// FB Controle/FB_PAlloc
(*
    ════════════════════════════════════════════════════════════════
    FB_PAlloc - Alocador de Potência Ativa (PRIORIDADE MÁXIMA)
    ════════════════════════════════════════════════════════════════
*)
FUNCTION_BLOCK FB_PAlloc
VAR_INPUT
    P_total_cmd_kW : REAL;          // Comando de P total (do FB_PI)
END_VAR

VAR_OUTPUT
    P_allocated_kW : REAL;          // ✅ ADICIONAR ESTA SAÍDA!
END_VAR

VAR
    i : UINT;
    P_target_i : REAL;
    P_actual_i : REAL;
    P_total_calc : REAL;
    proportion : REAL;
END_VAR


P_total_calc := 0.0;

FOR i := 1 TO Global.NMAXINVERSORES DO     
    
    IF GVL_Persis.InvActivePower[i] > 0.0 THEN
        
        // Proporção do inversor
        proportion := GVL_Persis.InvActivePower[i] / Global.InstalledPower;
        
        // P proporcional
        P_target_i := P_total_cmd_kW * proportion;
        
        // Limita apenas pela nominal (ignora S_max por enquanto)
        P_actual_i := MIN(P_target_i, GVL_Persis.InvActivePower[i]);
        
        // Armazena P
        Global.P_inv_kW[i] := P_actual_i;
        
        // Setpoint percentual
        IF GVL_Persis.InvActivePower[i] > 0.0 THEN
            Global.P_inv_Percent[i] := (P_actual_i / GVL_Persis.InvActivePower[i]) * 100.0;
        ELSE
            Global.P_inv_Percent[i] := 0.0;
        END_IF
        
        P_total_calc := P_total_calc + P_actual_i;
        
    ELSE
        Global.P_inv_kW[i] := 0.0;
        Global.P_inv_Percent[i] := 0.0;
    END_IF
    
END_FOR

// ✅ ATUALIZA SAÍDA
P_allocated_kW := P_total_calc;

END_FUNCTION_BLOCK

// FB Controle/FB_PI
FUNCTION_BLOCK FB_PI
VAR_INPUT
    setpoint    : REAL;         		// Setpoint desejado
    feedback    : REAL;         		// Medição atual (feedback)
    Kp          : REAL;         		// Ganho proporcional
    Ki          : REAL;         		// Ganho integral
    OutMax      : REAL;         		// Limite superior de saída
    OutMin      : REAL;         		// Limite inferior de saída
    CycleTime   : REAL;         		// Tempo de ciclo (s)
    RampUp      : REAL := 1.0E+6;  		//  Rampa de subida (unidade/s). Default = sem limite
    RampDown    : REAL := 1.0E+6;  		//  Rampa de descida (unidade/s). Default = sem limite
    Deadband    : REAL := 0.0;          //  deadband em kW (já convertido de %)
    bReset      : BOOL := FALSE;        //  reset do PI
END_VAR

VAR_OUTPUT
    u           : REAL;         		// Saída do controlador
    erro        : REAL;         		// Erro atual (setpoint - feedback)
    bSaturated  : BOOL;         		// TRUE = saída saturada
END_VAR

VAR
    integ           : REAL := 0.0;      // Integral acumulada
    LastOut         : REAL := 0.0;
    erroAtual       : REAL;             // Erro no ciclo atual
    u_prop          : REAL;             // Componente proporcional
    u_raw           : REAL;             // Saída antes da saturação
    u_limited       : REAL;         	// Saída após saturação, antes da rampa
    delta           : REAL;         	// Variação desejada
    delta_max       : REAL;         	// Variação máxima permitida
    primeiro_ciclo  : BOOL := TRUE;     // Flag de primeira execução
    sinal_saturacao : INT;              // +1: saturado max, -1: saturado min, 0: não saturado
END_VAR


// ════════════════════════════════════════════════════════════════
// Reset explícito
// ════════════════════════════════════════════════════════════════
IF bReset THEN
    integ := 0.0;
    LastOut := 0.0;
    u := 0.0;
    bSaturated := FALSE;
    primeiro_ciclo := TRUE;
    RETURN;
END_IF

// ════════════════════════════════════════════════════════════════
// Inicialização suave na primeira execução
// ════════════════════════════════════════════════════════════════
IF primeiro_ciclo THEN
    integ := 0.0;
    primeiro_ciclo := FALSE;
    
    // Se quiser inicializar LastOut com valor atual do medidor:
    // LastOut := feedback;  // Opcional: evita salto inicial
END_IF

// ════════════════════════════════════════════════════════════════
// Cálculo do Erro + Deadband
// ════════════════════════════════════════════════════════════════
erroAtual := setpoint - feedback;

// ✅ Deadband
IF ABS(erroAtual) < Deadband THEN
    erroAtual := 0.0;
END_IF

erro := erroAtual;  // Saída para diagnóstico

// ════════════════════════════════════════════════════════════════
// Componente Proporcional
// ════════════════════════════════════════════════════════════════
u_prop := Kp * erroAtual;

// ════════════════════════════════════════════════════════════════
// Saída Raw (P + I + LastOut)
// ══════════════════════════════════════════���═════════════════════
u_prop := Kp * erroAtual;
u_raw := u_prop + integ;

// ════════════════════════════════════════════════════════════════
// Saturação
// ════════════════════════════════════════════════════════════════
IF u_raw > OutMax THEN
    u_limited := OutMax;
    bSaturated := TRUE;
    sinal_saturacao := 1;
ELSIF u_raw < OutMin THEN
    u_limited := OutMin;
    bSaturated := TRUE;
    sinal_saturacao := -1;
ELSE
    u_limited := u_raw;
    bSaturated := FALSE;
    sinal_saturacao := 0;
END_IF

// ════════════════════════════════════════���═══════════════════════
// Rate Limiter (Rampa)
// ════════════════════════════════════════════════════════════════
delta := u_limited - LastOut;

IF delta > 0.0 THEN
    delta_max := RampUp * CycleTime;
    IF delta > delta_max THEN
        u := LastOut + delta_max;
    ELSE
        u := u_limited;
    END_IF
ELSIF delta < 0.0 THEN
    delta_max := RampDown * CycleTime;
    IF ABS(delta) > delta_max THEN
        u := LastOut - delta_max;
    ELSE
        u := u_limited;
    END_IF
ELSE
    u := u_limited;
END_IF
// ════════════════════════════════════════════════════════════════
// Anti-windup Melhorado (Conditional Integration)
// ════════════════════════════════════════════════════════════════
// Regras:
// 1. NÃO saturado → acumula normalmente
// 2. Saturado MAS erro na direção oposta → permite desacumular
// 3. Saturado E erro na mesma direção → freeze (não acumula)

IF NOT bSaturated THEN
    // Caso 1: Normal - acumula integral
    integ := integ + (Ki * erroAtual * CycleTime);
    
ELSIF (sinal_saturacao = 1 AND erroAtual < 0.0) OR (sinal_saturacao = -1 AND erroAtual > 0.0) THEN
    // Caso 2: Saturado MAS erro está tentando sair da saturação
    // Permite acumular para ajudar a desaturar
    integ := integ + (Ki * erroAtual * CycleTime);
    
ELSE
    // Caso 3: Saturado E erro empurrando mais para saturação
    // NÃO acumula (freeze integral)
    // integ permanece inalterado
END_IF

// ════════════════════════════════════════════════════════════════
// Atualiza LastOut
// ════════════════════════════════════════════════════════════════
LastOut := u;

END_FUNCTION_BLOCK

// FB Controle/FB_Diagnostico
(*
    ════════════════════════════════════════════════════════════════
    FB_Diagnostico - Diagnóstico de Fator de Potência
    ════════════════════════════════════════════════════════════════
    
    Gera diagnóstico completo do sistema de compensação de PF,
    incluindo alarmes, recomendações e estatísticas.
    
    ═══���════════════════════════════════════════════════════════════
*)

FUNCTION_BLOCK FB_Diagnostico
VAR_INPUT
    P_allocated_kW : REAL;
    Q_commanded_kvar : REAL;
    Q_allocated_kvar : REAL;
    Q_capacity_kvar : REAL;
    PF_measured : REAL;
    PF_achieved : REAL;
    bQ_limited : BOOL;
END_VAR

VAR
    Q_deficit : REAL;
    Q_deficit_pct : REAL;
    S_total_avail : REAL;
    S_total_used : REAL;
    bank_size : REAL;
    bank_size_int : DINT;  // ✅ DINT (não INT)
END_VAR

// ════════════════════════════════════════════════════════════════
// 1. ARMAZENA VALORES BÁSICOS
// ════════════════════════════════════════════════════════════════

Global.P_generated_kW := P_allocated_kW;
Global.P_allocated_kW := P_allocated_kW;
Global.Q_commanded_kvar := Q_commanded_kvar;
Global.Q_allocated_kvar := Q_allocated_kvar;
Global.Q_available_kvar := Q_capacity_kvar;
Global.PF_measured := PF_measured;
Global.PF_achieved := PF_achieved;

// Q medido (do ponto de conexão)
Global.Q_measured_kvar := Global.Qt;  // Já convertido em kvar pelo FB_AjustaLeitura

// ════════════════════════════════════════════════════════════════
// 2. CALCULA DÉFICIT DE Q
// ════════════════════════════════════════════════════════════════

Q_deficit := Q_commanded_kvar - Q_allocated_kvar;
Global.Q_deficit_kvar := Q_deficit;

// Déficit percentual
IF ABS(Q_commanded_kvar) > 0.1 THEN
    Q_deficit_pct := (ABS(Q_deficit) / ABS(Q_commanded_kvar)) * 100.0;
ELSE
    Q_deficit_pct := 0.0;
END_IF
Global.Q_deficit_percent := Q_deficit_pct;

// ════════════════════════════════════════════════════════════════
// 3. CALCULA UTILIZAÇÃO DE S
// ════════════════════════════════════════════════════════════════

// S total disponível
S_total_avail := Global.InstalledSmax;
Global.S_total_available_kVA := S_total_avail;

// S total usado
S_total_used := SQRT((P_allocated_kW * P_allocated_kW) + (Q_allocated_kvar * Q_allocated_kvar));
Global.S_total_used_kVA := S_total_used;

// Utilização percentual
IF S_total_avail > 0.0 THEN
    Global.S_utilization_pct := (S_total_used / S_total_avail) * 100.0;
ELSE
    Global.S_utilization_pct := 0.0;
END_IF

// ════════════════════════════════════════════════════════════════
// 4. CALCULA UTILIZAÇÃO DE Q
// ════════════════════════════════════════════════════════════════

Global.Q_capacity_total_kvar := Q_capacity_kvar;

IF Q_capacity_kvar > 0.0 THEN
    Global.Q_utilization_pct := (ABS(Q_allocated_kvar) / Q_capacity_kvar) * 100.0;
ELSE
    Global.Q_utilization_pct := 0.0;
END_IF

// ════════════════════════════════════════════════════════════════
// 5. CALCULA TAMANHO DE BANCO DE CAPACITORES
// ════════════════════════════════════════════════════════════════

IF Q_deficit > 0.1 THEN
    // Adiciona 10% de margem
    bank_size := ABS(Q_deficit) * 1.1;
	bank_size := DINT_TO_REAL(TRUNC(bank_size / 5.0) + 1) * 5.0;
    Global.Capacitor_bank_size_kvar := bank_size;
    Global.Capacitor_bank_recommended := TRUE;
ELSE
    Global.Capacitor_bank_size_kvar := 0.0;
    Global.Capacitor_bank_recommended := FALSE;
END_IF

// ════════════════════════════════════════════════════════════════
// 6. DETERMINA STATUS DE PF
// ════════════════════════════════════════════════════════════════

IF PF_achieved >= Global.PF_target THEN
    Global.PF_OK := TRUE;
    Global.PFErro := FALSE;
    Global.PF_alarm_code := 0;  // OK
    Global.PF_alarm_message := 'Fator de Potencia OK';
ELSE
    Global.PF_OK := FALSE;
    
    IF bQ_limited THEN
        Global.PFErro := TRUE;
        
        // Classifica severidade
        IF Q_deficit_pct > 20.0 THEN
            Global.PF_alarm_code := 2;  // Crítico
            Global.PF_alarm_message := 'CRITICO: Limite de Q atingido - Banco de capacitores necessario';
        ELSE
            Global.PF_alarm_code := 1;  // Aviso
            Global.PF_alarm_message := 'AVISO: Limite de Q atingido - Considerar banco de capacitores';
        END_IF
    ELSE
        // PF < 0.92 mas não por limite de Q (transitório)
        Global.PFErro := FALSE;
        Global.PF_alarm_code := 1;
        Global.PF_alarm_message := 'PF abaixo do alvo - Sistema compensando';
    END_IF
END_IF

// ════════════════════════════════════════════════════════════════
// 7. ATUALIZA HISTÓRICO (OPCIONAL - implementar com timers)
// ════════════════════════════════════════════════════════════════

// Atualiza PF mínimo
IF PF_achieved < Global.PF_min_24h THEN
    Global.PF_min_24h := PF_achieved;
END_IF

// Atualiza déficit máximo
IF Q_deficit > Global.Q_deficit_max_24h THEN
    Global.Q_deficit_max_24h := Q_deficit;
END_IF

// Conta alarmes (incrementar quando alarme dispara pela primeira vez)
// (Implementar com edge detection)

END_FUNCTION_BLOCK

// FB Controle/FB_PowerController
(*
    ════════════════════════════════════════════════════════════════
    FB_PowerController - Controlador de Potência Ativa
    ════════════════════════════════════════════════════════════════
    
    Responsabilidade:
    - Calcular comando de P (PI + Safety Margin + Limites de Fase)
    - Encapsular toda lógica relacionada a potência ativa
    
    Pipeline:
    1. PI → P_cmd_raw
    2. Safety Margin → P_cmd_with_margin
    3. Limitador de Fase → P_cmd_limited
    
    ════════════════════════════════════════════════════════════════
*)
FUNCTION_BLOCK FB_PowerController
VAR_INPUT
    ExportLimit_kW : REAL;      // Do scheduler (kW)
    Feedback_kW : REAL;         // Leitura do medidor (kW)
    bReset : BOOL;              // Reset do PI
END_VAR

VAR_OUTPUT
    P_cmd_kW : REAL;            // Comando final (kW)
    bSaturated : BOOL;          // PI saturado
    bPhase_limited : BOOL;      // Limitado por fase
    sLimited_phase : STRING;    // Qual fase limitou
    Margin_applied_kW : REAL;   // Margem aplicada (telemetria)
	EffectiveExportLimit_kW : REAL;
END_VAR

VAR
    // Sub-blocos
    fbPI : FB_PI;
    fbSafetyMargin : FB_SafetyMargin;
    fbFLimiter : FB_FLimiter;
	fbDroop : FB_DroopP;
    
    // Variáveis internas
    P_setpoint : REAL;
    P_cmd_raw : REAL;
    P_cmd_with_margin : REAL;
	lastInstalledPower : REAL := -1.0;
	
	// Droop
    P_error_kW : REAL;
    P_droop_kW : REAL;
	
    P_droop_max_kW : REAL;
    P_cmd_sum : REAL;
	
	// ✅ Deadband em kW (convertido de %)
	Deadband_P_kW     : REAL;
    Droop_Deadband_kW : REAL;
END_VAR

// ────────────────────────────────────────────────────────────────
// ETAPA 1: CONTROLADOR PI
// ────────────────────────────────────────────────────────────────

// Setpoint negativo (exportação)
P_setpoint := -ABS(ExportLimit_kW);

// Erro (kW)
P_error_kW := Feedback_kW - P_setpoint;

// Converte deadband (%) para kW (mínimo 1 kW)
// Recalcula apenas se InstalledPower mudou
IF lastInstalledPower <> Global.InstalledPower THEN
    Deadband_P_kW := MAX(1.0, Global.InstalledPower * (GVL_Persis.Deadband_P / 100.0));
    Droop_Deadband_kW := MAX(1.0, Global.InstalledPower * (GVL_Persis.Deadband_Droop / 100.0));
	Deadband_P_kW := MIN(20.0, MAX(1.0, Global.InstalledPower * (GVL_Persis.Deadband_P / 100.0)));
	Droop_Deadband_kW := MIN(20.0, MAX(1.0, Global.InstalledPower * (GVL_Persis.Deadband_Droop / 100.0)));		
    lastInstalledPower := Global.InstalledPower;
END_IF

// Limite máximo do droop (fração da potência instalada)
P_droop_max_kW := GVL_Persis.Droop_Max * Global.InstalledPower;

// Calcula droop
fbDroop(
    Enable      := GVL_Persis.Droop_Enable,
    bReset      := bReset,                 
    Error_kW    := P_error_kW,
    K_droop     := GVL_Persis.K_Droop,
    Deadband_kW := Droop_Deadband_kW,
    P_max_kW    := P_droop_max_kW
);

P_droop_kW := fbDroop.P_droop_kW;

// PI de potência ativa
fbPI(
    setpoint    := P_error_kW,
    feedback    := 0.0,
    Kp          := GVL_Persis.Kp_P,
    Ki          := GVL_Persis.Ki_P,
    OutMax      := Global.InstalledPower,
    OutMin      := 0.0,
    CycleTime   := Global.ControlCycle,
	RampUp      := GVL_Persis.RampUp_P,     
    RampDown    := GVL_Persis.RampDown_P,    
    Deadband    := Deadband_P_kW,
	bReset      := bReset          
);

// Soma droop + PI
P_cmd_sum := P_droop_kW + fbPI.u;

// Comando bruto (segue fluxo normal)
P_cmd_raw := P_cmd_sum;
IF P_cmd_raw < 0.0 THEN
    P_cmd_raw := 0.0;
ELSIF P_cmd_raw > Global.InstalledPower THEN
    P_cmd_raw := Global.InstalledPower;
END_IF
bSaturated := fbPI.bSaturated;

// ─────────────────────────────────────────���──────────────────────
// ETAPA 2: SAFETY MARGIN
// ────────────────────────────────────────────────────────────────

fbSafetyMargin(
    P_cmd_raw_kW := P_cmd_raw,
    Margin_pct := GVL_Persis.SafetyMargin_pct,
    TC_Power_kW := GVL_Persis.TC_Power_kW
);

P_cmd_with_margin := fbSafetyMargin.P_cmd_adjusted_kW;
Margin_applied_kW := fbSafetyMargin.Margin_applied_kW;  // ✅ Telemetria
EffectiveExportLimit_kW := P_setpoint + Margin_applied_kW;
// ────────────────────────────────────────────────────────────────
// ETAPA 3: LIMITADOR DE FASE
// ────────────────────────────────────────────────────────────────

fbFLimiter(
    P_cmd_in := P_cmd_with_margin,
    PowerMode := GVL_Persis.PowerMode
);

P_cmd_kW := fbFLimiter.P_cmd_out;
bPhase_limited := fbFLimiter.bPhase_limited;
sLimited_phase := fbFLimiter.sLimited_phase;

// ────────────────────────────────────────────────────────────────
// PROTEÇÃO FINAL: Potência Instalada
// ────────────────────────────────────────────────────────────────

IF P_cmd_kW > Global.InstalledPower THEN
    P_cmd_kW := Global.InstalledPower;
    bSaturated := TRUE;
END_IF

END_FUNCTION_BLOCK

// FB Controle/FB_SafetyMargin
(*
    ════════════════════════════════════════════════════════════════
    FB_SafetyMargin - Margem de Segurança para Correção de TC
    ════════════════════════════════════════════════════════════════
    
    Função:
    - Aplica margem de segurança para compensar erro de TC em baixas correntes
    - Desloca setpoint para lado da importação (garante não exportar)
    
    Exemplo:
    - P_cmd = 100 kW
    - TC_Power = 329 kW
    - Margin = 3%
    - SafetyMargin = 3% × 329 = 9.87 kW
    - P_adjusted = 100 - 9.87 = 90.13 kW
    ════════════════════════════════════════════════════════════════
*)
FUNCTION_BLOCK FB_SafetyMargin
VAR_INPUT
    P_cmd_raw_kW : REAL;        // Comando sem margem
    Margin_pct : REAL;          // Percentual (ex: 3.0)
    TC_Power_kW : REAL;         // Potência do TC
END_VAR

VAR_OUTPUT
    P_cmd_adjusted_kW : REAL;   // Comando com margem
    Margin_applied_kW : REAL;   // Margem aplicada (para telemetria)
END_VAR

VAR
    SafetyMargin_kW : REAL;
END_VAR

// ════════════════════════════════════════════════════════════════
// IMPLEMENTAÇÃO
// ════════════════════════════════════════════════════════════════
// 1. Proteção: se TC não configurado, não aplica margem
IF TC_Power_kW <= 0.0 THEN
    P_cmd_adjusted_kW := P_cmd_raw_kW;
    Margin_applied_kW := 0.0;
    RETURN;
END_IF

// 2. Calcula margem em kW
SafetyMargin_kW := (Margin_pct / 100.0) * TC_Power_kW;

// 3. Aplica margem (reduz comando)
P_cmd_adjusted_kW := P_cmd_raw_kW - SafetyMargin_kW;

// 4. Limita para não ficar negativo
IF P_cmd_adjusted_kW < 0.0 THEN
    P_cmd_adjusted_kW := 0.0;
END_IF

// 5. Armazena margem aplicada (para HMI)
Margin_applied_kW := SafetyMargin_kW;

END_FUNCTION_BLOCK

// FB Controle/FB_FLimiter
(*
    FB_FLimiter - Limitador por Fase
    
    Função:
    - Verifica se o comando causaria EXPORTAÇÃO excessiva em alguma fase
    - Se fase está IMPORTANDO: ignora (não há problema)
    - Se fase está EXPORTANDO: verifica se comando excederia limite
    
    Lógica:
    1. Calcula P futuro por fase = P_atual + (P_cmd / 3)
    2. Para cada fase EXPORTANDO (P < 0):
       - Verifica se P_futuro < P_phase_limit (mais exportação que permitido)
       - Se sim, calcula comando máximo para essa fase
    3. Usa o MENOR comando máximo entre as fases
    
    Convenção de sinais:
    - P > 0: Importação
    - P < 0: Exportação
    - MaxExportLimit: VALOR POSITIVO na agenda (ex: 90 kW)
    - P_phase_limit: NEGATIVO internamente (ex: -30 kW)
	    
    Exemplo:
    - Agenda: MaxExportLimit = 90 kW (sem sinal)
    - Internamente: P_phase_limit = -90/3 = -30 kW por fase
    - Se Pa = -25 kW (exportando 25 kW)
    - Se P_cmd = -18 kW (quer aumentar exportação)
    - P_future_A = -25 + (-18/3) = -31 kW → EXCEDE -30 kW → LIMITA
*)

FUNCTION_BLOCK FB_FLimiter
VAR_INPUT
    P_cmd_in : REAL;                // Comando de P calculado pelo PI (kW)
    PowerMode : UINT;               // 0=Total, 1=Por fase, 2=Ambos
END_VAR

VAR_OUTPUT
    P_cmd_out : REAL;               // Comando de P limitado por fase (kW)
    bPhase_limited : BOOL;          // TRUE = alguma fase limitou
	sLimited_phase : STRING;        // Qual fase limitou: 'A', 'B', 'C', 'AB', etc.
END_VAR

VAR
    P_cmd_per_phase : REAL;         // Comando adicional por fase (kW)
    P_future_A : REAL;              // P futuro na fase A após aplicar comando (kW)
    P_future_B : REAL;              // P futuro na fase B após aplicar comando (kW)
    P_future_C : REAL;              // P futuro na fase C após aplicar comando (kW)
    P_phase_limit : REAL;           // Limite de exportação por fase (kW negativo)
    P_max_cmd_A : REAL;             // Comando máximo permitido para fase A (kW)
    P_max_cmd_B : REAL;             // Comando máximo permitido para fase B (kW)
    P_max_cmd_C : REAL;             // Comando máximo permitido para fase C (kW)
    P_max_cmd_total : REAL;         // Comando máximo total permitido (kW)
	NO_LIMIT : REAL;                // Constante para "sem limite"
    bLimitA : BOOL;                 // Fase A está limitando
    bLimitB : BOOL;                 // Fase B está limitando
    bLimitC : BOOL;                 // Fase C está limitando
END_VAR

// Comando adicional por fase (distribuído equilibradamente)
P_cmd_per_phase := P_cmd_in / 3.0;

// Limite de exportação por fase
// Se MaxExportLimit = -90 kW, então por fase = -30 kW
P_phase_limit := -ABS(Global.MaxExportLimit) / 3.0;

// ════════════════════════════════════════════════════════════════
// ════════════════════════════════════════════════════════════════
// Inicialização
// ════════════════════════════════════════════════════════════════
NO_LIMIT := Global.InstalledPower * 10.0;  // Valor grande, mas realista
sLimited_phase := '';
bLimitA := FALSE;
bLimitB := FALSE;
bLimitC := FALSE;

// ════════════════════════════════════════════════════════════════
// Se PowerMode = 0, não verifica fase
// ════════════════════════════════════════════════════════════════
IF PowerMode = 0 THEN
    P_cmd_out := P_cmd_in;
    bPhase_limited := FALSE;
    RETURN;
END_IF

// ════════════════════════════════════════════════════════════════
// Proteção: Se InstalledPower não configurado
// ════════════════════════════════════════════════════════════════
IF Global.InstalledPower <= 0.0 THEN
    P_cmd_out := 0.0;
    bPhase_limited := TRUE;
    sLimited_phase := 'ERROR: InstalledPower=0';
    RETURN;
END_IF

// ════════════════════════════════════════════════════════════════
// Calcula P futuro em cada fase após aplicar comando
// ════════════════════════════════════════════════════════════════
P_future_A := Global.Pa + P_cmd_per_phase;
P_future_B := Global.Pb + P_cmd_per_phase;
P_future_C := Global.Pc + P_cmd_per_phase;

// ════════════════════════════════════════════════════════════════
// Verifica FASE A
// ════════════════════════════════════════════════════════════════
IF P_future_A < 0.0 THEN
    // Fase A estará EXPORTANDO após aplicar comando
    
    IF P_future_A < P_phase_limit THEN
        // Excederia o limite de exportação!
        // Calcula quanto PODE aumentar exportação sem exceder:
        // P_max_per_phase = P_limit - P_atual
        // P_max_total = P_max_per_phase * 3
        P_max_cmd_A := (P_phase_limit - Global.Pa) * 3.0;
        bLimitA := TRUE;
    ELSE
        // Dentro do limite: sem restrição
        P_max_cmd_A := NO_LIMIT;
    END_IF
    
ELSE
    // Fase A estará IMPORTANDO: sem problema
    P_max_cmd_A := NO_LIMIT;
END_IF

// ════════════════════════════════════════════════════════════════
// Verifica FASE B
// ════════════════════════════════════════════════════════════════
IF P_future_B < 0.0 THEN
    // Fase B estará EXPORTANDO
    
    IF P_future_B < P_phase_limit THEN
        P_max_cmd_B := (P_phase_limit - Global.Pb) * 3.0;
        bLimitB := TRUE;
    ELSE
        P_max_cmd_B := NO_LIMIT;
    END_IF
    
ELSE
    // Fase B estará IMPORTANDO
    P_max_cmd_B := NO_LIMIT;
END_IF

// ════════════════════════════════════════════════════════════════
// Verifica FASE C
// ════════════════════════════════════════════════════════════════
IF P_future_C < 0.0 THEN
    // Fase C estará EXPORTANDO
    
    IF P_future_C < P_phase_limit THEN
        P_max_cmd_C := (P_phase_limit - Global.Pc) * 3.0;
        bLimitC := TRUE;
    ELSE
        P_max_cmd_C := NO_LIMIT;
    END_IF
    
ELSE
    // Fase C estará IMPORTANDO
    P_max_cmd_C := NO_LIMIT;
END_IF

// ════════════════════════════════════════════════════════════════
// Aplica o MENOR limite (fase mais restritiva)
// ════════════════════════════════════════════════════════════════
P_max_cmd_total := MIN(P_max_cmd_A, MIN(P_max_cmd_B, P_max_cmd_C));

// ════════════════════════════════════════════════════════════════
// Verifica se houve limitação
// ════════════════════════════════════════════════════════════════
IF P_cmd_in > P_max_cmd_total THEN
    P_cmd_out := P_max_cmd_total;
    bPhase_limited := TRUE;
    
    // Identifica qual(is) fase(s) limitou
    IF bLimitA THEN sLimited_phase := CONCAT(sLimited_phase, 'A'); END_IF
    IF bLimitB THEN sLimited_phase := CONCAT(sLimited_phase, 'B'); END_IF
    IF bLimitC THEN sLimited_phase := CONCAT(sLimited_phase, 'C'); END_IF
    
ELSE
    P_cmd_out := P_cmd_in;
    bPhase_limited := FALSE;
    sLimited_phase := '';
END_IF

END_FUNCTION_BLOCK

// FB Controle/FB_DroopP
(*
    FB_DroopP - Droop para Potência Ativa
    Gera um comando base proporcional ao erro de potência.
    Uso: antes do PI (PI corrige residual).
*)
FUNCTION_BLOCK FB_DroopP
VAR_INPUT
    Enable        : BOOL;   // Habilita droop
    bReset        : BOOL;   // Reset do droop
    Error_kW      : REAL;   // Erro (Setpoint - Feedback)
    K_droop       : REAL;   // Ganho droop (kW/kW)
    Deadband_kW   : REAL;   // Zona morta
    P_max_kW      : REAL;   // Limite absoluto do droop (kW)
END_VAR

VAR_OUTPUT
    P_droop_kW    : REAL;   // Saída do droop (kW)
END_VAR

VAR
    P_cmd : REAL;
    erro  : REAL;
END_VAR

// ──────────────────────────────────��───────────────────────────
// Reset
// ──────────────────────────────────────────────────────────────
IF bReset THEN
    P_droop_kW := 0.0;
    RETURN;
END_IF

// ──────────────────────────────────────────────────────────────
// Lógica do droop
// ──────────────────────────────────────────────────────────────
IF NOT Enable THEN
    P_droop_kW := 0.0;
    RETURN;
END_IF

// Aplica deadband ao erro
erro := Error_kW;
IF ABS(erro) < Deadband_kW THEN
    erro := 0.0;
END_IF

P_cmd := K_droop * erro;

// Limite absoluto
IF P_cmd > P_max_kW THEN
    P_cmd := P_max_kW;
ELSIF P_cmd < -P_max_kW THEN
    P_cmd := -P_max_kW;
END_IF

P_droop_kW := P_cmd;

END_FUNCTION_BLOCK

// FB Leitura/FB_ReadMedidor
FUNCTION_BLOCK FB_ReadMedidor

VAR_INPUT
    Execute 				: BOOL;                 // habilita leitura
END_VAR

VAR_OUTPUT
    result 					: E_ModbusResult;      		 // resultado
    bDadosOK				: BOOL:= FALSE;  // Dados aprovados
	bPoucosErros			: BOOL:= TRUE;  // Inicialmente sem erros
END_VAR

VAR
	fbAlarmes				: FB_Alarmes;		 		// converte códigos de erros em mensagens texto
	fbChannel       		: ModbusChannel;
	fbValidaDadosRele		: FB_ValidaDadosRele;	
	
    state 					: (TRIG, WAIT) := TRIG;
	tonTimer				: TON;
	tTimeout				: TIME := T#250MS;			// tempo de leitura do medidor é cerca de 200 ms
END_VAR

// ============================================================
// Máquina de estados de leitura do medidor
// ============================================================

// estado default por ciclo
result := E_ModbusResult.BUSY;

// se não habilitado, não executa
IF NOT Execute THEN
    result := E_ModbusResult.END;
    Global.trigMedidor100 := FALSE;
	state := TRIG;
    RETURN;
END_IF

tonTimer(IN := (state = WAIT), PT := tTimeout);

CASE state OF

    TRIG:
        Global.trigMedidor100 := TRUE;      // trigger rising edge
        state := WAIT;

    WAIT:
        IF Global.pMedidor100^.xDone THEN
            Global.trigMedidor100 := FALSE;
            state := TRIG;
          	result := E_ModbusResult.DONE;
			fbValidaDadosRele();
			bDadosOK:=fbValidaDadosRele.bDadosOK;
			bPoucosErros:=fbValidaDadosRele.bPoucosErros;
			
        ELSIF Global.pMedidor100^.xError THEN
				fbChannel(Slave := Global.pMedidor100^,iChannelIndex := 0);
				fbAlarmes(codigo := fbChannel.ModbusError,tError:=TO_UDINT(SysTimeRtcGet(Global.Result)));
				state:= TRIG;
				Global.trigMedidor100:=FALSE;
          		result := E_ModbusResult.ERRO;
				
		ELSIF tonTimer.Q THEN
				fbAlarmes(codigo := 16#B2,tError:=TO_UDINT(SysTimeRtcGet(Global.Result)));
				state:= TRIG;
				Global.trigMedidor100:=FALSE;	
				result := E_ModbusResult.TIMEOUT;
		END_IF	

END_CASE

END_FUNCTION_BLOCK

// FB Leitura/FB_ValidaDadosRele
(*═════════════════════════════════════════════════════════════════════
 FB_ValidaMedicao
 
 Valida medições do medidor trifásico via Modbus, aplica filtro
 passa-baixa e verifica consistência física das grandezas.
 
 ENTRADAS:
 - (nenhuma - lê de valorLido.WordArray via Modbus)
 
 SAÍDAS:
 - bDadosOK: TRUE se medições são válidas
 - bPoucosErros: TRUE se < 5 erros consecutivos
 - diagnosticCode: Código de falha (0 = OK)
 
 LÓGICA:
 1. Conversão de escalas (Modbus → unidades físicas)
 2. Validação de ranges individuais
 3. Validação cruzada (Pt vs soma, PF vs P/S)
 4. Detecção de congelamento 
 5. Filtro passa-baixa exponencial (SOMENTE se validação OK)
 6. Atualização de variáveis globais (SOMENTE se validação OK)
 7. Janela de erros (5 consecutivos = FAIL_SAFE)
═════════════════════════════════════════════════════════════════════*)
FUNCTION_BLOCK FB_ValidaDadosRele

VAR_OUTPUT
    bDadosOK		: BOOL 	:= FALSE;  // Dados aprovados
	bPoucosErros	: BOOL  := TRUE;  // Inicialmente sem erros
    diagnosticCode 	: WORD;            // Código de falha
END_VAR

VAR
	valorLido		: UN_Rele;
	Ua    	    	: REAL := 0.0; // 2006H - Tensão de fase A x 0,1 V
	Ub    	    	: REAL := 0.0; // 2008H - Tensão de fase B x 0,1 V
	Uc    	    	: REAL := 0.0; // 200AH - Tensão de fase C x 0,1 V
	
	Ia    	    	: REAL := 0.0; // 200CH - Corrente de fase A x 0,001 A 
	Ib    	    	: REAL := 0.0; // 200EH - Corrente de fase B x 0,001 A
	Ic    	    	: REAL := 0.0; // 2010H - Corrente de fase C x 0,001 A
	
	Pt    	    	: REAL := 0.0; // 2012H - Potencia ativa combinada x 0,1 W
	Pa    	    	: REAL := 0.0; // 2014H - Potencia ativa fase A x 0,1 W
	Pb    	    	: REAL := 0.0; // 2016H - Potencia ativa fase B x 0,1 W
	Pc    	   		: REAL := 0.0; // 2018H - Potencia ativa fase C x 0,1 W	
		
	Qt    	    	: REAL := 0.0; // 201AH - Potencia reativa combinada x 0,1 var
	Qa    	    	: REAL := 0.0; // 201CH - Potencia reativa fase A x 0,1 var
	Qb    	    	: REAL := 0.0; // 201EH - Potencia reativa fase B x 0,1 var
	Qc    	    	: REAL := 0.0; // 2020H - Potencia reativa fase C x 0,1 var

	PFt    	    	: REAL := 0.0; // 202AH - Fator de potência combinado (número positivo: indutivo, número negativo: capacitivo) (x  0,001)
	PFa    	    	: REAL := 0.0; // 202CH - Fator de potência de fase A (número positivo: indutivo, número negativo: capacitivo)  (×0,001)
	PFb    	    	: REAL := 0.0; // 202EH - Fator de potência de fase B (número positivo: indutivo, número negativo: capacitivo)  (×0,001)
	PFc    	    	: REAL := 0.0; // 2030H - Fator de potência de fase C (número positivo: indutivo, número negativo: capacitivo)  (×0,001)
	
	// Limites físicos (ajustar conforme instalação)
    PFMIN 			: REAL := 0.5;
    PFMAX 			: REAL := 1.0;
	
	// variaveis auxiliares
    bRangeError 	: BOOL := FALSE;            // Fora de faixa
	nErrors 		: UINT := 0;
	SomaP			: REAL;
	SomaQ 			: REAL;
	Calculado 		: REAL;
	Tolerancia  	: REAL :=0.05;
	Pt_last 		: REAL := 0.0;
    frozen_count 	: UINT := 0;
	FREEZE_THRESHOLD: UINT := 10;  		// 10 ciclos
	bFirstRun		: BOOL :=TRUE;
	Pt_filt 		: REAL :=0;
    Qt_filt 		: REAL :=0;
    PFt_filt 		: REAL :=0;
END_VAR

// ═══════════════════════════════════════════════════════════════
// 1. RESET DE ESTADO
// ═══════════════════════════════════════════════════════════════

bRangeError := FALSE;
diagnosticCode := 0;

// ═══════════════════════════════════════════════════════════════
// 2. CONVERSÃO DE ESCALAS
// ═══════════════════════════════════════════════════════════════
Ua  := valorLido.EmReal.Ua * 0.1;				// em Volts
Ub  := valorLido.EmReal.Ub * 0.1;				// em Volts
Uc  := valorLido.EmReal.Uc * 0.1;				// em Volts

Ia  := valorLido.EmReal.Ia * 0.001;				// em Amperes
Ib  := valorLido.EmReal.Ib * 0.001;				// em Amperes
Ic  := valorLido.EmReal.Ic * 0.001;				// em Amperes

Pt  := valorLido.EmReal.Pt *0.0001;				// kW
Pa  := valorLido.EmReal.Pa *0.0001;				// kW
Pb  := valorLido.EmReal.Pb *0.0001;				// kW
Pc  := valorLido.EmReal.Pc *0.0001;				// kW

Qt  := valorLido.EmReal.Qt *0.0001;				// kvar
Qa  := valorLido.EmReal.Qa *0.0001;				// kvar
Qb  := valorLido.EmReal.Qb *0.0001;				// kvar
Qc  := valorLido.EmReal.Qc *0.0001;				// xkvar

PFt := valorLido.EmReal.PFt *0.001;	
PFa := valorLido.EmReal.PFa *0.001;
PFb := valorLido.EmReal.PFb *0.001;
PFc := valorLido.EmReal.PFc *0.001;

// ═══════════════════════════════════════════════════════════════
// 3. VALIDAÇÃO DE RANGES (SEM RETURN)
// ═══════════════════════════════════════════════════════════════
// validação de tensões
IF (Ua < GVL_Persis.VMIN) OR (Ua > GVL_Persis.VMAX) THEN
    bRangeError := TRUE;
    diagnosticCode := 16#A101;  				// Erro de tensão fase A
END_IF
IF (Ub < GVL_Persis.VMIN) OR (Ub > GVL_Persis.VMAX) THEN
    bRangeError := TRUE;
    diagnosticCode := 16#A102;  				// Erro de tensão fase B
END_IF
IF (Uc < GVL_Persis.VMIN) OR (Uc > GVL_Persis.VMAX) THEN
    bRangeError := TRUE;
    diagnosticCode := 16#A103;  				// Erro de tensão fase B
END_IF

// validação de correntes
IF (ABS(Ia) > GVL_Persis.IMAX) THEN
    bRangeError := TRUE;
    diagnosticCode := 16#A201;  				// Erro de corrente fase A
END_IF
IF (ABS(Ib) > GVL_Persis.IMAX) THEN
    bRangeError := TRUE;
    diagnosticCode := 16#A202;  				// Erro de corrente fase B
END_IF
IF (ABS(Ic) > GVL_Persis.IMAX) THEN
    bRangeError := TRUE;
    diagnosticCode := 16#A203;  				// Erro de corrente fase C
END_IF

// validação de potencias ativas
IF (ABS(Pt) > GVL_Persis.PMAX) THEN
    bRangeError := TRUE;
    diagnosticCode := 16#A301;  				// Erro de potência total
END_IF
IF (ABS(Pa) > GVL_Persis.PMAX) THEN
    bRangeError := TRUE;
    diagnosticCode := 16#A302;  				// Erro de potência Pa
END_IF
IF (ABS(Pb) > GVL_Persis.PMAX) THEN
    bRangeError := TRUE;
    diagnosticCode := 16#A303;  				// Erro de potência Pb
END_IF
IF (ABS(Pc) > GVL_Persis.PMAX) THEN
    bRangeError := TRUE;
    diagnosticCode := 16#A304;    				// Erro de potência Pc
END_IF

// validação de potencias reativas
IF (ABS(Qt) > GVL_Persis.QMAX) THEN
    bRangeError := TRUE;
    diagnosticCode := 16#A401;  				// Erro de potência Qt
END_IF
IF (ABS(Qa) > GVL_Persis.QMAX) THEN
    bRangeError := TRUE;
    diagnosticCode := 16#A402;  				// Erro de potência Qa
END_IF
IF (ABS(Qb) > GVL_Persis.QMAX) THEN
    bRangeError := TRUE;
    diagnosticCode := 16#A403;  				// Erro de potência Qb
END_IF
IF (ABS(Qc) > GVL_Persis.QMAX) THEN
    bRangeError := TRUE;
    diagnosticCode := 16#A404;  				// Erro de potência Qc
END_IF
	
// validação do fator das potencias
	
IF (ABS(PFt) < PFMIN) OR (ABS(PFt) >PFMAX)  THEN
    bRangeError := TRUE;
    diagnosticCode := 16#A501;  				// Erro de PFt
END_IF
IF (ABS(PFa) < PFMIN) OR (ABS(PFa) >PFMAX)  THEN
    bRangeError := TRUE;
    diagnosticCode := 16#A502;  				// Erro de PFa
END_IF
IF (ABS(PFb) < PFMIN) OR (ABS(PFb) >PFMAX)  THEN
    bRangeError := TRUE;
    diagnosticCode := 16#A503;  				// Erro de PFb
END_IF
IF (ABS(PFc) < PFMIN) OR (ABS(PFc) >PFMAX)  THEN
    bRangeError := TRUE;
    diagnosticCode := 16#A504;  				// Erro de PFc
END_IF

// ═══════════════════════════════════════════════════════════════
// 4. VALIDAÇÃO CRUZADA (SÓ SE NÃO HOUVER ERRO AINDA)
// ═══════════════════════════════════════════════════════════════

IF NOT bRangeError THEN
	// Só valida se Pa significativo (ex: > 1 kW)
	IF ABS(Pa) > 1.0 THEN
		Calculado := Ua * Ia * PFa / 1000;
		IF ABS(Pa - Calculado) > (ABS(Pa) * Tolerancia) THEN  // ✅ Usa Pa, não Calculado
			bRangeError := TRUE;
			diagnosticCode := 16#A601;
		END_IF
	END_IF
	
	// Repetir para Pb e Pc
	IF ABS(Pb) > 1.0 THEN
		Calculado := Ub * Ib * PFb / 1000;
		IF ABS(Pb - Calculado) > (ABS(Pb) * Tolerancia) THEN
			bRangeError := TRUE;
			diagnosticCode := 16#A602;
		END_IF
	END_IF
	
	IF ABS(Pc) > 1.0 THEN
		Calculado := Uc * Ic * PFc / 1000;
		IF ABS(Pc - Calculado) > (ABS(Pc) * Tolerancia) THEN
			bRangeError := TRUE;
			diagnosticCode := 16#A603;
		END_IF
	END_IF
	// Pt = Pa + Pb + Pc
	SomaP := Pa + Pb + Pc;
	IF ABS(Pt) > 1.0 THEN  // ✅ Só valida se significativo
		IF ABS(Pt - SomaP) > (ABS(Pt) * Tolerancia) THEN  // ✅ Usa Pt
			bRangeError := TRUE;
			diagnosticCode := 16#A604;
		END_IF
	END_IF
	
	// FPt com base nas potencias ativas e reativas
	SomaQ:=Qa + Qb + Qc;
	Calculado := SQRT((SomaP * SomaP)+ (SomaQ * SomaQ));
	IF Calculado > 10 THEN 									// 1 kva
		Calculado := SomaP / Calculado;
		IF ABS(PFt - Calculado) > 0.05 THEN
			bRangeError := TRUE;
			diagnosticCode := 16#A605;  
		END_IF
	END_IF
END_IF;

// ═══════════════════════════════════════════════════════════════
// 5. DETECÇÃO DE CONGELAMENTO (OPCIONAL)
// ═══════════════════════════════════════════════════════════════
IF NOT bRangeError THEN
	IF ABS(Pt - Pt_last) < 1.0 THEN  // < 1 kW de variação
		frozen_count := frozen_count + 1;
	ELSE
		frozen_count := 0;
	END_IF
	
	IF frozen_count > FREEZE_THRESHOLD THEN
		bRangeError := TRUE;
		diagnosticCode := 16#A900;
	END_IF
END_IF

Pt_last := Pt;
// ═══════════════════════════════════════════════════════════════
// 6. TRATAMENTO FINAL DE ERRO/SUCESSO
// ═══════════════════════════════════════════════════════==══════
IF bRangeError THEN
	
    nErrors := MIN(nErrors + 1, 10);  // Clamp em 10
    bDadosOK := FALSE;  // Dado atual é inválido
    
    IF nErrors >= 5 THEN
        bPoucosErros := FALSE;  // 🚨 Degradação crítica
    ELSE
        bPoucosErros := TRUE;   // ⚠️ Ainda tolerável (1-4 erros)
    END_IF
    // ❌ NÃO atualiza variáveis globais (mantém último valor válido)
    // ❌ NÃO reseta filtro (preserva estado anterior)  
ELSE
	// 1. Decrementa contador de erros (recuperação gradual)
    IF nErrors > 0 THEN
        nErrors := nErrors - 1;
    END_IF
    
    bDadosOK := TRUE;
    bPoucosErros := TRUE;
    diagnosticCode := 0;
	
    // 2. FILTRO PASSA-BAIXA (Suavização de Medição)
    // ─────────────────────────────────────────────────────────
    IF bFirstRun THEN
        Pt_filt := Pt;
        Qt_filt := Qt;
        PFt_filt := PFt;
        bFirstRun := FALSE;
    ELSE
		// Filtro exponencial: y[n] = α·x[n] + (1-α)·y[n-1]
        // ALPHA configurável (ex: 0.25 → ~3s para 95% do valor)
        Pt_filt := GVL_Persis.ALPHA * Pt + (1.0 - GVL_Persis.ALPHA) * Pt_filt;
        Qt_filt := GVL_Persis.ALPHA * Qt + (1.0 - GVL_Persis.ALPHA) * Qt_filt;
        PFt_filt := GVL_Persis.ALPHA * PFt + (1.0 - GVL_Persis.ALPHA) * PFt_filt;
    END_IF
	
	// 3. ATUALIZAÇÃO DE VARIÁVEIS GLOBAIS
    // ──────────────────────────────────────────────────────────
	Global.Ua  := Ua;				// em Volts
	Global.Ub  := Ub;				// em Volts
	Global.Uc  := Uc;				// em Volts
	
	Global.Ia  := Ia;				// em Amperes
	Global.Ib  := Ib;				// em Amperes
	Global.Ic  := Ic;				// em Amperes
	
	// Potência Ativa (FILTRADA para controle)
	Global.Pt  := Pt_filt;			// kW
	Global.Pa  := Pa;				// kW
	Global.Pb  := Pb;				// kW
	Global.Pc  := Pc;				// kW
	
	// Potência Reativa (FILTRADA para controle de PF)
	Global.Qt  := Qt_filt;			// kvar
	Global.Qa  := Qa;				// kvar
	Global.Qb  := Qb;				// kvar
	Global.Qc  := Qc;				// kvar
    
    // Fator de Potência (FILTRADO para controle)
	Global.PFt := PFt_filt;				
	Global.PFa := PFa;
	Global.PFb := PFb;
	Global.PFc := PFc;

END_IF

END_FUNCTION_BLOCK

// FB Escrita/FB_WriteInv
FUNCTION_BLOCK FB_WriteInv

VAR_INPUT
    Execute     : BOOL;
    InvIndex    : UINT;
END_VAR

VAR_IN_OUT
    trigInv     : BOOL;                    // ex.: Global.trigInvCOM100[i]
    pSlave      : ModbusSlaveComPort;      // ex.: Global.pInversores100[i]^
END_VAR

VAR_OUTPUT
    result      : E_ModbusResult;
END_VAR

VAR
    fbAlarmes   : FB_Alarmes;
    fbChannel   : ModbusChannel;
    state       : (TRIG, WAIT) := TRIG;
    tonTimer    : TON;
    tTimeout    : TIME := T#150MS;
END_VAR

// ============================================================
// Máquina de estados de escrita em inversores
// ============================================================

// estado default por ciclo
result := E_ModbusResult.BUSY;

// bloqueio por Execute
IF NOT Execute THEN
    trigInv := FALSE;
    state := TRIG;
    result := E_ModbusResult.END;
    RETURN;
END_IF

tonTimer(IN := (state = WAIT), PT := tTimeout);

CASE state OF

    TRIG:
        trigInv := TRUE;
        state := WAIT;

    WAIT:
       IF pSlave.xDone THEN
            trigInv := FALSE;
            state := TRIG;
            result := E_ModbusResult.DONE;
			
		
      	ELSIF pSlave.xError THEN
            fbChannel(Slave := pSlave, iChannelIndex := 0);
            fbAlarmes(codigo := fbChannel.ModbusError,tError := TO_UDINT(SysTimeRtcGet(Global.Result)));
            state := TRIG;
            trigInv := FALSE;
            result := E_ModbusResult.ERRO;
			
      	ELSIF tonTimer.Q THEN
            fbAlarmes(codigo := 16#B2,tError := TO_UDINT(SysTimeRtcGet(Global.Result)));
            state := TRIG;
            trigInv := FALSE;
            result := E_ModbusResult.TIMEOUT;
        END_IF
END_CASE

END_FUNCTION_BLOCK

// Eventos/FB_EventLog
// ════════════════════════════════════════════════════════════════════
// FB_EventLog — Buffer rotativo de eventos em NVRAM
// ════════════════════════════════════════════════════════════════════
// Plataforma: WAGO CC100 / CODESYS V3.5 SP21 Patch 4
//
// RESPONSABILIDADES:
//   1. Armazenar eventos em ring buffer RETAIN (sobrevive a power-cycle)
//   2. Limitar a 1 escrita por chamada (proteção de NVRAM)
//   3. Fornecer último evento e contadores para HMI
//   4. Permitir leitura indexada para exportação/diagnóstico
//
// GARANTIAS:
//   - Nunca estoura array (índice clamped por MOD)
//   - Nunca aloca memória dinâmica
//   - Tempo de execução O(1) por chamada (sem loops)
//   - Não usa STRING em runtime
//
// USO:
//   fbEventLog.LogEvent(
//       eCode      := E_EventCode.CRIT_HARD_LIMIT_15S,
//       bRaised    := TRUE,
//       rParam1    := Global.Pt,
//       rParam2    := REAL#-500.0,   // limite violado
//       uMachState := UINT_TO_UINT(MachineState)
//   );
// ════════════════════════════════════════════════════════════════════
FUNCTION_BLOCK FB_EventLog
VAR RETAIN
    // ── Ring buffer persistente ──
    aBuffer         : ARRAY[0..(GVL_EventLog.MAX_EVENT_ENTRIES - 1)] OF ST_EventEntry;
    nHead           : UINT := 0;            // Próxima posição de escrita
    bWrapped        : BOOL := FALSE;        // TRUE = buffer já deu pelo menos uma volta completa
    nTotalLogged    : UDINT := 0;           // Contador total desde último factory reset (para telemetria)
END_VAR
VAR
    // ── Saídas para HMI / lógica externa (recalculadas a cada LogEvent) ──
    stLastEvent     : ST_EventEntry;        // Cópia do último evento registrado
    nCount          : UINT := 0;            // Quantas entradas válidas existem no buffer
    bOverflow       : BOOL := FALSE;        // Sinaliza que eventos antigos foram sobrescritos
END_VAR

METHOD Clear
VAR
    i : UINT;
END_VAR
FOR i := 0 TO (GVL_EventLog.MAX_EVENT_ENTRIES - 1) DO
    aBuffer[i].tTimestamp   := 0;
    aBuffer[i].eCode        := E_EventCode.EVT_NONE;
    aBuffer[i].bRaised      := FALSE;
    aBuffer[i].rParam1      := 0.0;
    aBuffer[i].rParam2      := 0.0;
    aBuffer[i].uMachState   := 0;
END_FOR

nHead := 0;
bWrapped := FALSE;
nTotalLogged := 0;
nCount := 0;
bOverflow := FALSE;

// Registra o próprio clear como primeiro evento do buffer limpo
// (para rastreabilidade — saber que houve reset intencional)
LogEvent(
    eCode       := E_EventCode.INFO_STARTUP_BEGIN,  // Reutiliza como "system reset"
    bRaised     := TRUE,
    rParam1     := 0.0,
    rParam2     := 0.0,
    uMachState  := 0
);
END_METHOD

// ════════════════════════════════════════════════════════════════════
// METHOD GetEvent — Lê evento por índice reverso (0 = mais recente)
// ════════════════════════════════════════════════════════════════════
// Para HMI: exibe os últimos N eventos em ordem cronológica reversa.
// Para exportação: itera de 0 a nCount-1.
//
// Retorna TRUE se o índice é válido, FALSE se fora do range.
// Quando retorna FALSE, stOut fica zerado (não retorna lixo).
// ════════════════════════════════════════════════════════════════════
METHOD GetEvent : BOOL
VAR_INPUT
    nReverseIndex   : UINT;     // 0 = mais recente, 1 = anterior, ...
END_VAR
VAR_OUTPUT
    stOut           : ST_EventEntry;
END_VAR
VAR
    nActualIdx      : UINT;
    nTemp           : INT;
END_VAR
// Validação de range
IF nReverseIndex >= nCount THEN
    // Índice fora do range — zera saída e retorna FALSE
    stOut.tTimestamp     := 0;
    stOut.eCode          := E_EventCode.EVT_NONE;
    stOut.bRaised        := FALSE;
    stOut.rParam1        := 0.0;
    stOut.rParam2        := 0.0;
    stOut.uMachState     := 0;
    GetEvent := FALSE;
    RETURN;
END_IF

// Calcula índice real no buffer circular
// nHead aponta para a PRÓXIMA posição de escrita.
// Último escrito = nHead - 1.
// Índice reverso N = nHead - 1 - N (com wrap-around).
nTemp := UINT_TO_INT(nHead) - 1 - UINT_TO_INT(nReverseIndex);
IF nTemp < 0 THEN
    nTemp := nTemp + UINT_TO_INT(GVL_EventLog.MAX_EVENT_ENTRIES);
END_IF
nActualIdx := INT_TO_UINT(nTemp);

stOut := aBuffer[nActualIdx];
GetEvent := TRUE;
END_METHOD

// ════════════════════════════════════════════════════════════════════
// METHOD LogEvent — Insere um evento no ring buffer
// ════════════════════════════════════════════════════════════════════
// Complexidade: O(1). Uma escrita de struct + incremento de ponteiro.
// Pode ser chamado de qualquer FB (ErrorManager, MainProgram, etc.)
//
// IMPORTANTE: Não chame mais de ~5 vezes por ciclo de scan (1s).
// Em cascata de falhas, o caller deve agregar — ex.: registrar
// apenas o primeiro erro de range por ciclo, não um por fase.
// ════════════════════════════════════════════════════════════════════
METHOD LogEvent
VAR_INPUT
    eCode           : E_EventCode;      // Código do evento
    bRaised         : BOOL;             // TRUE = raise, FALSE = clear
    rParam1         : REAL := 0.0;      // Contexto #1 (opcional)
    rParam2         : REAL := 0.0;      // Contexto #2 (opcional)
    uMachState      : UINT := 0;        // Estado da máquina (opcional)
END_VAR
VAR
    tNow            : UDINT;
    result          : RTS_IEC_RESULT;
END_VAR
// ── 1. Obter timestamp ──
// SysTimeRtcGet retorna epoch UTC em segundos.
// Se RTC falhar (result <> 0), registra timestamp = 0.
// O evento AINDA É REGISTRADO — melhor ter evento sem hora
// do que perder evento crítico por falha de RTC.
tNow := SysTimeRtcGet(pResult := ADR(result));
IF result <> 0 THEN
    tNow := 0;  // Sinaliza "RTC indisponível" — não descarta o evento
END_IF

// ── 2. Escrever no buffer ──
// nHead já é a posição correta (calculada no final do último LogEvent)
aBuffer[nHead].tTimestamp   := tNow;
aBuffer[nHead].eCode        := eCode;
aBuffer[nHead].bRaised      := bRaised;
aBuffer[nHead].rParam1      := rParam1;
aBuffer[nHead].rParam2      := rParam2;
aBuffer[nHead].uMachState   := uMachState;

// ── 3. Atualizar cópia do último evento (para HMI) ──
stLastEvent := aBuffer[nHead];

// ── 4. Avançar ponteiro circular ──
nHead := (nHead + 1) MOD GVL_EventLog.MAX_EVENT_ENTRIES;

// ── 5. Detectar wrap-around ──
IF nHead = 0 THEN
    bWrapped := TRUE;
END_IF

// ── 6. Atualizar contadores ──
nTotalLogged := nTotalLogged + 1;

// nCount = quantas entradas válidas existem
IF bWrapped THEN
    nCount := GVL_EventLog.MAX_EVENT_ENTRIES;
    bOverflow := TRUE;
ELSE
    nCount := nHead;    // Antes do wrap, nHead = número de entradas escritas
    bOverflow := FALSE;
END_IF
END_METHOD

END_FUNCTION_BLOCK

// FB da IHM/FB_EventDisplay
// ════════════════════════════════════════════════════════════════════
// FB_EventDisplay — Prepara eventos do ring buffer para exibição na IHM
// ════════════════════════════════════════════════════════════════════
// A IHM não navega o ring buffer diretamente. Este FB expõe
// N linhas "flat" prontas para bind em Text Fields.
//
// Suporta paginação: nPageOffset controla qual "página" exibir.
//   Página 0 = eventos mais recentes
//   Página 1 = próximos DISPLAY_LINES eventos, etc.
//
// Chamado sob demanda (quando operador abre a tela de histórico),
// NÃO a cada ciclo.
// ════════════════════════════════════════════════════════════════════
FUNCTION_BLOCK FB_EventDisplay

VAR_INPUT
    pEventLog       : REFERENCE TO FB_EventLog;     // Referência ao ring buffer
    bRefresh        : BOOL;                         // Pulso = atualiza dados
    nPageOffset     : UINT := 0;                    // Página (0 = mais recente)
END_VAR

VAR_OUTPUT
    nTotalEvents    : UINT;                         // Total de eventos no buffer
    nTotalPages     : UINT;                         // Total de páginas disponíveis
    nCurrentPage    : UINT;                         // Página atual (0-based)
END_VAR

VAR CONSTANT
    DISPLAY_LINES   : UINT := 10;                   // Linhas visíveis na tela
END_VAR

VAR
    // ── Dados "flat" para a IHM (cada linha = 1 evento) ──
    asTimestamp      : ARRAY[0..9] OF STRING(20);   // 'DD/MM HH:MM:SS'
    asMessage        : ARRAY[0..9] OF STRING(60);   // Mensagem legível
    asParam1         : ARRAY[0..9] OF STRING(12);   // Valor contexto 1
    asParam2         : ARRAY[0..9] OF STRING(12);   // Valor contexto 2
    asSeverity       : ARRAY[0..9] OF STRING(8);    // 'INFO'/'WARN'/'ALARM'/'CRIT'
    asRaised         : ARRAY[0..9] OF STRING(5);    // 'RAISE' / 'CLEAR'
    abLineValid      : ARRAY[0..9] OF BOOL;         // TRUE = linha tem dados
	asCodeHex        : ARRAY[0..9] OF STRING(8);    // ex: '16#8700'

    // Auxiliares
    i               : UINT;
    nStartIdx       : UINT;
    stEvt           : ST_EventEntry;
    bOK             : BOOL;
    rTrigRefresh    : R_TRIG;
END_VAR

// ════════════════════════════════════════════════════════════════════
// Corpo do FB_EventDisplay — executa quando bRefresh tem borda de subida
// ════════════════════════════════════════════════════════════════════
rTrigRefresh(CLK := bRefresh);

IF rTrigRefresh.Q THEN

    // Total de eventos e páginas
    nTotalEvents := pEventLog.nCount;
    IF nTotalEvents > 0 THEN
        nTotalPages := ((nTotalEvents - 1) / DISPLAY_LINES) + 1;
    ELSE
        nTotalPages := 0;
    END_IF

    // Clamp página
    IF nPageOffset >= nTotalPages THEN
        nPageOffset := 0;
    END_IF
    nCurrentPage := nPageOffset;

    // Índice inicial no ring buffer (reverso)
    nStartIdx := nPageOffset * DISPLAY_LINES;

    // Preencher linhas
    FOR i := 0 TO (DISPLAY_LINES - 1) DO

        bOK := pEventLog.GetEvent(
            nReverseIndex := nStartIdx + i,
            stOut => stEvt
        );

        IF bOK THEN
            abLineValid[i] := TRUE;

            // Timestamp → string legível
            asTimestamp[i] := FC_EpochToString(stEvt.tTimestamp);

            // Código → mensagem
            asMessage[i] := FC_EventCodeToString(stEvt.eCode);

            // Severidade (extraída do nibble alto do código)
            asSeverity[i] := FC_SeverityToString(stEvt.eCode);

            // Raise/Clear
            IF stEvt.bRaised THEN
                asRaised[i] := 'RAISE';
            ELSE
                asRaised[i] := 'CLEAR';
            END_IF

            // Parâmetros numéricos formatados
            asParam1[i] := REAL_TO_STRING(stEvt.rParam1);
            asParam2[i] := REAL_TO_STRING(stEvt.rParam2);
			asCodeHex[i] := FC_UIntToHex16Sharp(TO_UINT(stEvt.eCode));
        ELSE
            // Linha vazia
            abLineValid[i]  := FALSE;
            asTimestamp[i]  := '';
            asMessage[i]    := '';
            asSeverity[i]   := '';
            asRaised[i]     := '';
            asParam1[i]     := '';
            asParam2[i]     := '';
			asCodeHex[i] 	:= '';
        END_IF

    END_FOR

END_IF

END_FUNCTION_BLOCK

// FB da IHM/FC_EpochToString
// ════════════════════════════════════════════════════════════════════
// FC_EpochToString — Converte UDINT epoch UTC para string legível
// ════════════════════════════════════════════════════════════════════
// Formato: 'DD/MM HH:MM:SS'
// Simplificação: usa SysTimeRtcConvertUtcToLocal + formatação manual
// Se tTimestamp = 0, retorna '-- sem RTC --'
// ════════════════════════════════════════════════════════════════════
FUNCTION FC_EpochToString : STRING(20)
VAR_INPUT
    tEpoch : UDINT;
END_VAR
VAR
    dtLocal     : DT;
    sTemp       : STRING(20);
    nDay        : UINT;
    nMonth      : UINT;
    nHour       : UINT;
    nMin        : UINT;
    nSec        : UINT;
END_VAR

IF tEpoch = 0 THEN
    FC_EpochToString := '-- sem RTC --';
    RETURN;
END_IF

// Converte epoch UDINT para DT (DATE_AND_TIME)
// DT no CODESYS V3 é segundos desde 01/01/1970 (mesmo que UDINT epoch)
dtLocal := UDINT_TO_DT(tEpoch);

// Extrai componentes usando funções padrão do SysTime / Util
// Nota: a implementação exata depende das libs disponíveis no target.
// Alternativa simples — usar DT_TO_STRING e truncar:
sTemp := DT_TO_STRING(dtLocal);

// DT_TO_STRING retorna formato 'DT#YYYY-MM-DD-HH:MM:SS'
// Extraímos apenas 'DD/MM HH:MM:SS' (14 chars)
FC_EpochToString := MID(sTemp, 2, 12);  // DD
FC_EpochToString := CONCAT(FC_EpochToString, '/');
FC_EpochToString := CONCAT(FC_EpochToString, MID(sTemp, 2, 9)); // MM
FC_EpochToString := CONCAT(FC_EpochToString, ' ');
FC_EpochToString := CONCAT(FC_EpochToString, MID(sTemp, 8, 15)); // HH:MM:SS

END_FUNCTION

// FB da IHM/FC_EventCodeToString
// ════════════════════════════════════════════════════════════════════
// FC_EventCodeToString — Mensagem legível para E_EventCode (PPC-GD)
// ════════════════════════════════════════════════════════════════════
// Uso: s := FC_EventCodeToString(E_EventCode.CRIT_HARD_LIMIT_15S);
// ════════════════════════════════════════════════════════════════════
FUNCTION FC_EventCodeToString : STRING(80)
VAR_INPUT
    eCode : E_EventCode;
END_VAR

CASE eCode OF
    // =============================================================
    // NONE
    // =============================================================
    E_EventCode.EVT_NONE:
        FC_EventCodeToString := '';

    // =============================================================
    // INFO (0x1xxx)
    // =============================================================
    // Startup (0x11xx)
    E_EventCode.INFO_STARTUP_BEGIN:
        FC_EventCodeToString := 'Startup: inicio';
    E_EventCode.INFO_SERIAL_COM_OK:
        FC_EventCodeToString := 'Startup: comunicacao serial OK';
    E_EventCode.INFO_RTC_OK:
        FC_EventCodeToString := 'Startup: RTC OK';
    E_EventCode.INFO_INVERTER_COUNT:
        FC_EventCodeToString := 'Startup: quantidade de inversores detectada';
    E_EventCode.INFO_INSTALLED_POWER:
        FC_EventCodeToString := 'Startup: potencia instalada OK';
    E_EventCode.INFO_K1_CONFIRMED:
        FC_EventCodeToString := 'Startup: K1 confirmado';
    E_EventCode.INFO_K2_CONFIRMED:
        FC_EventCodeToString := 'Startup: K2 confirmado';
    E_EventCode.INFO_STARTUP_DONE:
        FC_EventCodeToString := 'Startup: concluido';

    // Medição / Operação (0x12xx)
    E_EventCode.INFO_MEDIDOR_READ_OK:
        FC_EventCodeToString := 'Medidor: leitura OK';
    E_EventCode.INFO_MEDIDOR_DATA_VALID:
        FC_EventCodeToString := 'Medidor: dados validos';
    E_EventCode.INFO_MEAS_RECOVERING:
        FC_EventCodeToString := 'Medicao: recuperando (erros reduzindo)';

    // Escrita inversores (0x13xx)
    E_EventCode.INFO_WRITE_INV_OK:
        FC_EventCodeToString := 'Inversores: escrita OK';

    // Scheduler (0x15xx)
    E_EventCode.INFO_SPECIAL_DATE_ACTIVE:
        FC_EventCodeToString := 'Scheduler: data especial ativa';
    E_EventCode.INFO_ZERO_GRID_MODE:
        FC_EventCodeToString := 'Scheduler: modo zero grid ativo';

    // Máquina de estados (0x16xx)
    E_EventCode.INFO_CYCLE_COMPLETE:
        FC_EventCodeToString := 'Ciclo: completo';
    E_EventCode.INFO_FAIL_RECOVERY:
        FC_EventCodeToString := 'FAIL: recuperacao automatica';
    E_EventCode.INFO_STATE_CHANGE:
        FC_EventCodeToString := 'Maquina de estados: mudanca de estado';

    // STOP/Reset (0x18xx)
    E_EventCode.INFO_STOP_K2_OPEN_CONFIRMED:
        FC_EventCodeToString := 'STOP: K2 aberto confirmado';
    E_EventCode.INFO_STOP_RESET_APPROVED:
        FC_EventCodeToString := 'STOP: reset aprovado';
    E_EventCode.INFO_STOP_RESET_WAITING:
        FC_EventCodeToString := 'STOP: aguardando reset';

    // =============================================================
    // WARNING (0x2xxx)
    // =============================================================
    // Startup
    E_EventCode.WARN_TC_POWER_NOT_SET:
        FC_EventCodeToString := 'Startup: TC Power nao configurado';
    E_EventCode.WARN_NO_INVERSORES_COM02:
        FC_EventCodeToString := 'Startup: nenhum inversor no COM2';

    // Medição
    E_EventCode.WARN_MEAS_USING_LAST_VALID:
        FC_EventCodeToString := 'Medicao: usando ultimo valor valido';
    E_EventCode.WARN_MEAS_CROSS_CHECK_PA:
        FC_EventCodeToString := 'Medicao: cross-check Pa falhou';
    E_EventCode.WARN_MEAS_CROSS_CHECK_PB:
        FC_EventCodeToString := 'Medicao: cross-check Pb falhou';
    E_EventCode.WARN_MEAS_CROSS_CHECK_PC:
        FC_EventCodeToString := 'Medicao: cross-check Pc falhou';
    E_EventCode.WARN_MEAS_CROSS_CHECK_PT_SUM:
        FC_EventCodeToString := 'Medicao: cross-check Pt != Pa+Pb+Pc';
    E_EventCode.WARN_MEAS_CROSS_CHECK_PF:
        FC_EventCodeToString := 'Medicao: cross-check PF falhou';
    E_EventCode.WARN_MEAS_ERROR_ISOLATED:
        FC_EventCodeToString := 'Medicao: erro isolado (toleravel)';

    // Comunicação inversores
    E_EventCode.WARN_WRITE_INV_ERROR:
        FC_EventCodeToString := 'Inversores: erro de escrita';
    E_EventCode.WARN_WRITE_INV_TIMEOUT:
        FC_EventCodeToString := 'Inversores: timeout de escrita';

    // Controle
    E_EventCode.WARN_P_ALLOC_SATURATED:
        FC_EventCodeToString := 'Controle: alocacao de P saturada';
    E_EventCode.WARN_Q_LIMITED_BY_SMAX:
        FC_EventCodeToString := 'Controle: Q limitado por Smax';
    E_EventCode.WARN_PF_BELOW_TARGET:
        FC_EventCodeToString := 'Controle: PF abaixo do alvo';
    E_EventCode.WARN_PF_NOT_ACHIEVABLE:
        FC_EventCodeToString := 'Controle: PF nao atingivel';
    E_EventCode.WARN_PI_P_SATURATED:
        FC_EventCodeToString := 'Controle: PI de P saturado';
    E_EventCode.WARN_PI_Q_SATURATED:
        FC_EventCodeToString := 'Controle: PI de Q saturado';
    E_EventCode.WARN_PHASE_LIMITED:
        FC_EventCodeToString := 'Controle: limitado por fase';

    // Ciclo / watchdog
    E_EventCode.WARN_SCAN_OVERRUN:
        FC_EventCodeToString := 'Sistema: scan overrun';

    // STOP/reset
    E_EventCode.WARN_STOP_RESET_DENIED:
        FC_EventCodeToString := 'STOP: reset negado';

    // =============================================================
    // ALARM (0x4xxx)
    // =============================================================
    // Medição — Range/Freeze
    E_EventCode.ALARM_MEAS_VOLTAGE_A_RANGE:
        FC_EventCodeToString := 'Medicao: tensao fase A fora de faixa';
    E_EventCode.ALARM_MEAS_VOLTAGE_B_RANGE:
        FC_EventCodeToString := 'Medicao: tensao fase B fora de faixa';
    E_EventCode.ALARM_MEAS_VOLTAGE_C_RANGE:
        FC_EventCodeToString := 'Medicao: tensao fase C fora de faixa';
    E_EventCode.ALARM_MEAS_CURRENT_A_RANGE:
        FC_EventCodeToString := 'Medicao: corrente fase A fora de faixa';
    E_EventCode.ALARM_MEAS_CURRENT_B_RANGE:
        FC_EventCodeToString := 'Medicao: corrente fase B fora de faixa';
    E_EventCode.ALARM_MEAS_CURRENT_C_RANGE:
        FC_EventCodeToString := 'Medicao: corrente fase C fora de faixa';
    E_EventCode.ALARM_MEAS_PT_RANGE:
        FC_EventCodeToString := 'Medicao: Pt fora de faixa';
    E_EventCode.ALARM_MEAS_PA_RANGE:
        FC_EventCodeToString := 'Medicao: Pa fora de faixa';
    E_EventCode.ALARM_MEAS_PB_RANGE:
        FC_EventCodeToString := 'Medicao: Pb fora de faixa';
    E_EventCode.ALARM_MEAS_PC_RANGE:
        FC_EventCodeToString := 'Medicao: Pc fora de faixa';
    E_EventCode.ALARM_MEAS_QT_RANGE:
        FC_EventCodeToString := 'Medicao: Qt fora de faixa';
    E_EventCode.ALARM_MEAS_QA_RANGE:
        FC_EventCodeToString := 'Medicao: Qa fora de faixa';
    E_EventCode.ALARM_MEAS_QB_RANGE:
        FC_EventCodeToString := 'Medicao: Qb fora de faixa';
    E_EventCode.ALARM_MEAS_QC_RANGE:
        FC_EventCodeToString := 'Medicao: Qc fora de faixa';
    E_EventCode.ALARM_MEAS_PFT_RANGE:
        FC_EventCodeToString := 'Medicao: PFt fora de faixa';
    E_EventCode.ALARM_MEAS_PFA_RANGE:
        FC_EventCodeToString := 'Medicao: PFa fora de faixa';
    E_EventCode.ALARM_MEAS_PFB_RANGE:
        FC_EventCodeToString := 'Medicao: PFb fora de faixa';
    E_EventCode.ALARM_MEAS_PFC_RANGE:
        FC_EventCodeToString := 'Medicao: PFc fora de faixa';
    E_EventCode.ALARM_MEAS_FROZEN:
        FC_EventCodeToString := 'Medicao: congelada (frozen)';

    // Comunicação medidor
    E_EventCode.ALARM_MEDIDOR_MODBUS_ERROR:
        FC_EventCodeToString := 'Medidor: erro Modbus';
    E_EventCode.ALARM_MEDIDOR_TIMEOUT:
        FC_EventCodeToString := 'Medidor: timeout';

    // Comunicação inversores (canal degradado)
    E_EventCode.ALARM_COM_CH1_DEGRADED:
        FC_EventCodeToString := 'Inversores: COM1 degradado';
    E_EventCode.ALARM_COM_CH2_DEGRADED:
        FC_EventCodeToString := 'Inversores: COM2 degradado';

    // =============================================================
    // CRITICAL (0x8xxx)
    // =============================================================
    // Startup
    E_EventCode.CRIT_SERIAL_INIT_FAILED:
        FC_EventCodeToString := 'Startup: falha init serial';
    E_EventCode.CRIT_RTC_FAILED:
        FC_EventCodeToString := 'Startup: falha RTC';
    E_EventCode.CRIT_NO_INSTALLED_POWER:
        FC_EventCodeToString := 'Startup: potencia instalada = 0';
    E_EventCode.CRIT_K1_TIMEOUT:
        FC_EventCodeToString := 'Startup: timeout K1';

    // Medição
    E_EventCode.CRIT_MEAS_PERSISTENT_FAIL:
        FC_EventCodeToString := 'Medicao: falha persistente';
    E_EventCode.CRIT_MEDIDOR_COM_FAIL:
        FC_EventCodeToString := 'Medidor: falha comunicacao';

    // Comunicação inversores
    E_EventCode.CRIT_COM_CHANNEL_FAIL:
        FC_EventCodeToString := 'Inversores: falha canal comunicacao';

    // Controle
    E_EventCode.CRIT_INSTALLED_POWER_ZERO:
        FC_EventCodeToString := 'Controle: potencia instalada zero';

    // Scheduler
    E_EventCode.CRIT_RTC_READ_FAIL:
        FC_EventCodeToString := 'Scheduler: falha leitura RTC';
    E_EventCode.CRIT_SCHEDULE_INDEX_INVALID:
        FC_EventCodeToString := 'Scheduler: indice invalido';

    // Watchdog
    E_EventCode.CRIT_SCAN_WATCHDOG:
        FC_EventCodeToString := 'Sistema: watchdog de scan';

    // Proteções normativas
    E_EventCode.CRIT_HARD_LIMIT_15S:
        FC_EventCodeToString := 'Protecao: HardLimit >15s';
    E_EventCode.CRIT_EXPORT_OVER_LPI_30S:
        FC_EventCodeToString := 'Protecao: Exportacao >LPI >30s';
    E_EventCode.CRIT_MEDIDOR_TIMEOUT_IN_FAIL:
        FC_EventCodeToString := 'Protecao: timeout medidor em FAIL';

    // STOP / Trip
    E_EventCode.CRIT_STOP_ENTRY:
        FC_EventCodeToString := 'STOP: entrada em STOP';
    E_EventCode.CRIT_K2_DID_NOT_OPEN:
        FC_EventCodeToString := 'STOP: K2 nao abriu';
    E_EventCode.CRIT_STATE_CORRUPTION:
        FC_EventCodeToString := 'Sistema: corrupcao de estado';

ELSE
    FC_EventCodeToString := 'Evento desconhecido';
END_CASE

END_FUNCTION

// FB da IHM/FC_SeverityToString
// ════════════════════════════════════════════════════════════════════
// FC_SeverityToString — Extrai severidade do nibble alto de E_EventCode
// ════════════════════════════════════════════════════════════════════
FUNCTION FC_SeverityToString : STRING(8)
VAR_INPUT
    eCode : E_EventCode;
END_VAR
VAR
    nHighNibble : UINT;
END_VAR

nHighNibble := (TO_UINT(eCode) AND 16#F000);

CASE nHighNibble OF
    16#1000: FC_SeverityToString := 'INFO';
    16#2000: FC_SeverityToString := 'WARN';
    16#4000: FC_SeverityToString := 'ALARM';
    16#8000: FC_SeverityToString := 'CRIT';
ELSE
    FC_SeverityToString := '???';
END_CASE

END_FUNCTION

// FB da IHM/FC_UIntToHex16Sharp
// ════════════════════════════════════════════════════════════════════
// FC_UIntToHex16Sharp — Formata UINT como '16#XXXX' (4 nibbles)
// Ex.: 16#8700 -> '16#8700'
// tentar usar UINT_TO_HEXSTR se o CODESYS aceitar
// ════════════════════════════════════════════════════════════════════
FUNCTION FC_UIntToHex16Sharp : STRING(7)
VAR_INPUT
    uValue : UINT;
END_VAR
VAR
    aHex   : STRING(16) := '0123456789ABCDEF';
    n0, n1, n2, n3 : UINT;
    sOut : STRING(7);
END_VAR

n3 := (uValue AND 16#000F);
n2 := (SHR(uValue, 4)  AND 16#000F);
n1 := (SHR(uValue, 8)  AND 16#000F);
n0 := (SHR(uValue, 12) AND 16#000F);

// Monta '16#' + 4 dígitos
sOut := '16#';
sOut := CONCAT(sOut, MID(aHex, n0 + 1, 1));
sOut := CONCAT(sOut, MID(aHex, n1 + 1, 1));
sOut := CONCAT(sOut, MID(aHex, n2 + 1, 1));
sOut := CONCAT(sOut, MID(aHex, n3 + 1, 1));

FC_UIntToHex16Sharp := sOut;

END_FUNCTION

// FB Leitura/FB_ValidaDadosMedidor
(*═════════════════════════════════════════════════════════════════════
 FB_ValidaMedicao
 
 Valida medições do medidor trifásico via Modbus, aplica filtro
 passa-baixa e verifica consistência física das grandezas.
 
 ENTRADAS:
 - (nenhuma - lê de valorLido.WordArray via Modbus)
 
 SAÍDAS:
 - bDadosOK: TRUE se medições são válidas
 - bPoucosErros: TRUE se < 5 erros consecutivos
 - diagnosticCode: Código de falha (0 = OK)
 
 LÓGICA:
 1. Conversão de escalas (Modbus → unidades físicas)
 2. Validação de ranges individuais
 3. Validação cruzada (Pt vs soma, PF vs P/S)
 4. Detecção de congelamento 
 5. Filtro passa-baixa exponencial (SOMENTE se validação OK)
 6. Atualização de variáveis globais (SOMENTE se validação OK)
 7. Janela de erros (5 consecutivos = FAIL_SAFE)
═════════════════════════════════════════════════════════════════════*)
FUNCTION_BLOCK FB_ValidaDadosMedidor

VAR_OUTPUT
    bDadosOK		: BOOL 	:= FALSE;  // Dados aprovados
	bPoucosErros	: BOOL  := TRUE;  // Inicialmente sem erros
    diagnosticCode 	: WORD;            // Código de falha
END_VAR

VAR
	valorLido		: UN_Rele;
	Ua    	    	: REAL := 0.0; // 2006H - Tensão de fase A x 0,1 V
	Ub    	    	: REAL := 0.0; // 2008H - Tensão de fase B x 0,1 V
	Uc    	    	: REAL := 0.0; // 200AH - Tensão de fase C x 0,1 V
	
	Ia    	    	: REAL := 0.0; // 200CH - Corrente de fase A x 0,001 A 
	Ib    	    	: REAL := 0.0; // 200EH - Corrente de fase B x 0,001 A
	Ic    	    	: REAL := 0.0; // 2010H - Corrente de fase C x 0,001 A
	
	Pt    	    	: REAL := 0.0; // 2012H - Potencia ativa combinada x 0,1 W
	Pa    	    	: REAL := 0.0; // 2014H - Potencia ativa fase A x 0,1 W
	Pb    	    	: REAL := 0.0; // 2016H - Potencia ativa fase B x 0,1 W
	Pc    	   		: REAL := 0.0; // 2018H - Potencia ativa fase C x 0,1 W	
		
	Qt    	    	: REAL := 0.0; // 201AH - Potencia reativa combinada x 0,1 var
	Qa    	    	: REAL := 0.0; // 201CH - Potencia reativa fase A x 0,1 var
	Qb    	    	: REAL := 0.0; // 201EH - Potencia reativa fase B x 0,1 var
	Qc    	    	: REAL := 0.0; // 2020H - Potencia reativa fase C x 0,1 var

	PFt    	    	: REAL := 0.0; // 202AH - Fator de potência combinado (número positivo: indutivo, número negativo: capacitivo) (x  0,001)
	PFa    	    	: REAL := 0.0; // 202CH - Fator de potência de fase A (número positivo: indutivo, número negativo: capacitivo)  (×0,001)
	PFb    	    	: REAL := 0.0; // 202EH - Fator de potência de fase B (número positivo: indutivo, número negativo: capacitivo)  (×0,001)
	PFc    	    	: REAL := 0.0; // 2030H - Fator de potência de fase C (número positivo: indutivo, número negativo: capacitivo)  (×0,001)
	
	// Limites físicos (ajustar conforme instalação)
    PFMIN 			: REAL := 0.5;
    PFMAX 			: REAL := 1.0;
	
	// variaveis auxiliares
    bRangeError 	: BOOL := FALSE;            // Fora de faixa
	nErrors 		: UINT := 0;
	SomaP			: REAL;
	SomaQ 			: REAL;
	Calculado 		: REAL;
	Tolerancia  	: REAL :=0.05;
	Pt_last 		: REAL := 0.0;
    frozen_count 	: UINT := 0;
	FREEZE_THRESHOLD: UINT := 10;  		// 10 ciclos
	bFirstRun		: BOOL :=TRUE;
	Pt_filt 		: REAL :=0;
    Qt_filt 		: REAL :=0;
    PFt_filt 		: REAL :=0;
END_VAR

// ═══════════════════════════════════════════════════════════════
// 1. RESET DE ESTADO
// ═══════════════════════════════════════════════════════════════

bRangeError := FALSE;
diagnosticCode := 0;

// ═══════════════════════════════════════════════════════════════
// 2. CONVERSÃO DE ESCALAS
// ═══════════════════════════════════════════════════════════════
Ua  := valorLido.EmReal.Ua * 0.1;				// em Volts
Ub  := valorLido.EmReal.Ub * 0.1;				// em Volts
Uc  := valorLido.EmReal.Uc * 0.1;				// em Volts

Ia  := valorLido.EmReal.Ia * 0.001;				// em Amperes
Ib  := valorLido.EmReal.Ib * 0.001;				// em Amperes
Ic  := valorLido.EmReal.Ic * 0.001;				// em Amperes

Pt  := valorLido.EmReal.Pt *0.0001;				// kW
Pa  := valorLido.EmReal.Pa *0.0001;				// kW
Pb  := valorLido.EmReal.Pb *0.0001;				// kW
Pc  := valorLido.EmReal.Pc *0.0001;				// kW

Qt  := valorLido.EmReal.Qt *0.0001;				// kvar
Qa  := valorLido.EmReal.Qa *0.0001;				// kvar
Qb  := valorLido.EmReal.Qb *0.0001;				// kvar
Qc  := valorLido.EmReal.Qc *0.0001;				// xkvar

PFt := valorLido.EmReal.PFt *0.001;	
PFa := valorLido.EmReal.PFa *0.001;
PFb := valorLido.EmReal.PFb *0.001;
PFc := valorLido.EmReal.PFc *0.001;

// ═══════════════════════════════════════════════════════════════
// 3. VALIDAÇÃO DE RANGES (SEM RETURN)
// ═══════════════════════════════════════════════════════════════
// validação de tensões
IF (Ua < GVL_Persis.VMIN) OR (Ua > GVL_Persis.VMAX) THEN
    bRangeError := TRUE;
    diagnosticCode := 16#A101;  				// Erro de tensão fase A
END_IF
IF (Ub < GVL_Persis.VMIN) OR (Ub > GVL_Persis.VMAX) THEN
    bRangeError := TRUE;
    diagnosticCode := 16#A102;  				// Erro de tensão fase B
END_IF
IF (Uc < GVL_Persis.VMIN) OR (Uc > GVL_Persis.VMAX) THEN
    bRangeError := TRUE;
    diagnosticCode := 16#A103;  				// Erro de tensão fase B
END_IF

// validação de correntes
IF (ABS(Ia) > GVL_Persis.IMAX) THEN
    bRangeError := TRUE;
    diagnosticCode := 16#A201;  				// Erro de corrente fase A
END_IF
IF (ABS(Ib) > GVL_Persis.IMAX) THEN
    bRangeError := TRUE;
    diagnosticCode := 16#A202;  				// Erro de corrente fase B
END_IF
IF (ABS(Ic) > GVL_Persis.IMAX) THEN
    bRangeError := TRUE;
    diagnosticCode := 16#A203;  				// Erro de corrente fase C
END_IF

// validação de potencias ativas
IF (ABS(Pt) > GVL_Persis.PMAX) THEN
    bRangeError := TRUE;
    diagnosticCode := 16#A301;  				// Erro de potência total
END_IF
IF (ABS(Pa) > GVL_Persis.PMAX) THEN
    bRangeError := TRUE;
    diagnosticCode := 16#A302;  				// Erro de potência Pa
END_IF
IF (ABS(Pb) > GVL_Persis.PMAX) THEN
    bRangeError := TRUE;
    diagnosticCode := 16#A303;  				// Erro de potência Pb
END_IF
IF (ABS(Pc) > GVL_Persis.PMAX) THEN
    bRangeError := TRUE;
    diagnosticCode := 16#A304;    				// Erro de potência Pc
END_IF

// validação de potencias reativas
IF (ABS(Qt) > GVL_Persis.QMAX) THEN
    bRangeError := TRUE;
    diagnosticCode := 16#A401;  				// Erro de potência Qt
END_IF
IF (ABS(Qa) > GVL_Persis.QMAX) THEN
    bRangeError := TRUE;
    diagnosticCode := 16#A402;  				// Erro de potência Qa
END_IF
IF (ABS(Qb) > GVL_Persis.QMAX) THEN
    bRangeError := TRUE;
    diagnosticCode := 16#A403;  				// Erro de potência Qb
END_IF
IF (ABS(Qc) > GVL_Persis.QMAX) THEN
    bRangeError := TRUE;
    diagnosticCode := 16#A404;  				// Erro de potência Qc
END_IF
	
// validação do fator das potencias
	
IF (ABS(PFt) < PFMIN) OR (ABS(PFt) >PFMAX)  THEN
    bRangeError := TRUE;
    diagnosticCode := 16#A501;  				// Erro de PFt
END_IF
IF (ABS(PFa) < PFMIN) OR (ABS(PFa) >PFMAX)  THEN
    bRangeError := TRUE;
    diagnosticCode := 16#A502;  				// Erro de PFa
END_IF
IF (ABS(PFb) < PFMIN) OR (ABS(PFb) >PFMAX)  THEN
    bRangeError := TRUE;
    diagnosticCode := 16#A503;  				// Erro de PFb
END_IF
IF (ABS(PFc) < PFMIN) OR (ABS(PFc) >PFMAX)  THEN
    bRangeError := TRUE;
    diagnosticCode := 16#A504;  				// Erro de PFc
END_IF

// ═══════════════════════════════════════════════════════════════
// 4. VALIDAÇÃO CRUZADA (SÓ SE NÃO HOUVER ERRO AINDA)
// ═══════════════════════════════════════════════════════════════

IF NOT bRangeError THEN
	// Só valida se Pa significativo (ex: > 1 kW)
	IF ABS(Pa) > 1.0 THEN
		Calculado := Ua * Ia * PFa / 1000;
		IF ABS(Pa - Calculado) > (ABS(Pa) * Tolerancia) THEN  // ✅ Usa Pa, não Calculado
			bRangeError := TRUE;
			diagnosticCode := 16#A601;
		END_IF
	END_IF
	
	// Repetir para Pb e Pc
	IF ABS(Pb) > 1.0 THEN
		Calculado := Ub * Ib * PFb / 1000;
		IF ABS(Pb - Calculado) > (ABS(Pb) * Tolerancia) THEN
			bRangeError := TRUE;
			diagnosticCode := 16#A602;
		END_IF
	END_IF
	
	IF ABS(Pc) > 1.0 THEN
		Calculado := Uc * Ic * PFc / 1000;
		IF ABS(Pc - Calculado) > (ABS(Pc) * Tolerancia) THEN
			bRangeError := TRUE;
			diagnosticCode := 16#A603;
		END_IF
	END_IF
	// Pt = Pa + Pb + Pc
	SomaP := Pa + Pb + Pc;
	IF ABS(Pt) > 1.0 THEN  // ✅ Só valida se significativo
		IF ABS(Pt - SomaP) > (ABS(Pt) * Tolerancia) THEN  // ✅ Usa Pt
			bRangeError := TRUE;
			diagnosticCode := 16#A604;
		END_IF
	END_IF
	
	// FPt com base nas potencias ativas e reativas
	SomaQ:=Qa + Qb + Qc;
	Calculado := SQRT((SomaP * SomaP)+ (SomaQ * SomaQ));
	IF Calculado > 10 THEN 									// 1 kva
		Calculado := SomaP / Calculado;
		IF ABS(PFt - Calculado) > 0.05 THEN
			bRangeError := TRUE;
			diagnosticCode := 16#A605;  
		END_IF
	END_IF
END_IF;

// ═══════════════════════════════════════════════════════════════
// 5. DETECÇÃO DE CONGELAMENTO (OPCIONAL)
// ═══════════════════════════════════════════════════════════════
IF NOT bRangeError THEN
	IF ABS(Pt - Pt_last) < 1.0 THEN  // < 1 kW de variação
		frozen_count := frozen_count + 1;
	ELSE
		frozen_count := 0;
	END_IF
	
	IF frozen_count > FREEZE_THRESHOLD THEN
		bRangeError := TRUE;
		diagnosticCode := 16#A900;
	END_IF
END_IF

Pt_last := Pt;
// ═══════════════════════════════════════════════════════════════
// 6. TRATAMENTO FINAL DE ERRO/SUCESSO
// ═══════════════════════════════════════════════════════==══════
IF bRangeError THEN
	
    nErrors := MIN(nErrors + 1, 10);  // Clamp em 10
    bDadosOK := FALSE;  // Dado atual é inválido
    
    IF nErrors >= 5 THEN
        bPoucosErros := FALSE;  // 🚨 Degradação crítica
    ELSE
        bPoucosErros := TRUE;   // ⚠️ Ainda tolerável (1-4 erros)
    END_IF    
    // ❌ NÃO atualiza variáveis globais (mantém último valor válido)
    // ❌ NÃO reseta filtro (preserva estado anterior)  
ELSE
	// 1. Decrementa contador de erros (recuperação gradual)
    IF nErrors > 0 THEN
        nErrors := nErrors - 1;
    END_IF
    
    bDadosOK := TRUE;
    bPoucosErros := TRUE;
    diagnosticCode := 0;
	
    // 2. FILTRO PASSA-BAIXA (Suavização de Medição)
    // ─────────────────────────────────────────────────────────
    IF bFirstRun THEN
        Pt_filt := Pt;
        Qt_filt := Qt;
        PFt_filt := PFt;
        bFirstRun := FALSE;
    ELSE
		// Filtro exponencial: y[n] = α·x[n] + (1-α)·y[n-1]
        // ALPHA configurável (ex: 0.25 → ~3s para 95% do valor)
        Pt_filt := GVL_Persis.ALPHA * Pt + (1.0 - GVL_Persis.ALPHA) * Pt_filt;
        Qt_filt := GVL_Persis.ALPHA * Qt + (1.0 - GVL_Persis.ALPHA) * Qt_filt;
        PFt_filt := GVL_Persis.ALPHA * PFt + (1.0 - GVL_Persis.ALPHA) * PFt_filt;
    END_IF
	
	// 3. ATUALIZAÇÃO DE VARIÁVEIS GLOBAIS
    // ──────────────────────────────────────────────────────────
	Global.Ua  := Ua;				// em Volts
	Global.Ub  := Ub;				// em Volts
	Global.Uc  := Uc;				// em Volts
	
	Global.Ia  := Ia;				// em Amperes
	Global.Ib  := Ib;				// em Amperes
	Global.Ic  := Ic;				// em Amperes
	
	// Potência Ativa (FILTRADA para controle)
	Global.Pt  := Pt_filt;			// kW
	Global.Pa  := Pa;				// kW
	Global.Pb  := Pb;				// kW
	Global.Pc  := Pc;				// kW
	
	// Potência Reativa (FILTRADA para controle de PF)
	Global.Qt  := Qt_filt;			// kvar
	Global.Qa  := Qa;				// kvar
	Global.Qb  := Qb;				// kvar
	Global.Qc  := Qc;				// kvar
    
    // Fator de Potência (FILTRADO para controle)
	Global.PFt := PFt_filt;				
	Global.PFa := PFa;
	Global.PFb := PFb;
	Global.PFc := PFc;

END_IF

END_FUNCTION_BLOCK

(* text list InverterComms (id | default)
   |  *)

(* text list Measurement (id | default)
   |  *)

(* text list Protection (id | default)
   |  *)

(* text list Startup (id | default)
  0 | 
   |  *)

(* text list StopTrip (id | default)
   |  *)

(* text list SystemWatchdog (id | default)
   |  *)
